# EPICS autosave request: autosave/galil_motors.req
$(P)$(M)_able
$(P)$(M)Direction
$(P)$(M)Offset
$(P)$(M)Resolution
$(P)$(M)_PCOF_SP
$(P)$(M)_ICOF_SP
$(P)$(M)_DCOF_SP
$(P)$(M)_ACCL_SP
$(P)$(M)_RDBD_SP
$(P)$(M)_VMAX_SP
$(P)$(M)_VELO_SP
$(P)$(M)_OFF_SP
$(P)$(M)_MRES_SP
$(P)$(M)_ERES_SP
$(P)$(M)_DIR_SP
$(P)$(M)_DMOV_SP
$(P)$(M)_SET_SP
$(P)$(M)_UEIP_SP
$(P)$(M)_SPMG_SP
$(P)$(M)_PREM_CMD
$(P)$(M)_POST_CMD
# $(P)$(M)_STOPGO_CMD
$(P)$(M)_VALOUT_SP
$(P)$(M).ACCL
$(P)$(M).ADEL
$(P)$(M).BACC
$(P)$(M).BDST
$(P)$(M).BVEL
$(P)$(M).CNEN
$(P)$(M).DCOF
$(P)$(M).DHLM
$(P)$(M).DINP
$(P)$(M).DIR
$(P)$(M).DLLM
$(P)$(M).DLY
$(P)$(M).DVAL
$(P)$(M).EGU
$(P)$(M).ERES
$(P)$(M).FOF
$(P)$(M).FOFF
$(P)$(M).FRAC
$(P)$(M).HHSV
$(P)$(M).HIGH
$(P)$(M).HIHI
$(P)$(M).HLM
$(P)$(M).HLSV
$(P)$(M).RDBL

$(P)$(M).HOMF
$(P)$(M).HOMR
$(P)$(M).HOPR
$(P)$(M).HSV
$(P)$(M).HVEL
$(P)$(M).ICOF
$(P)$(M).IGSET
$(P)$(M).INIT
$(P)$(M).JAR
$(P)$(M).JOGR
$(P)$(M).JOGF
$(P)$(M).JVEL
$(P)$(M).LLM
$(P)$(M).LLSV
$(P)$(M).LOCK
$(P)$(M).LOLO
$(P)$(M).LOPR
$(P)$(M).LOW
$(P)$(M).LSV
$(P)$(M).MDEL
$(P)$(M).NTM
$(P)$(M).NTMF
$(P)$(M).OFF
$(P)$(M).OMSL
$(P)$(M).OUT
$(P)$(M).PCOF
$(P)$(M).POST
$(P)$(M).PREC
$(P)$(M).PREM
$(P)$(M).RDBD
$(P)$(M).RINP
$(P)$(M).RLV
$(P)$(M).RMOD
$(P)$(M).RRES
$(P)$(M).RTRY
$(P)$(M).RVAL
$(P)$(M).S
$(P)$(M).SBAK
$(P)$(M).SBAS
$(P)$(M).SET
$(P)$(M).SMAX
$(P)$(M).SPMG
$(P)$(M).SREV
$(P)$(M).SSET
$(P)$(M).STOO
$(P)$(M).STOP
$(P)$(M).STUP
$(P)$(M).SUSE
$(P)$(M).SYNC
$(P)$(M).TWF
$(P)$(M).TWR
$(P)$(M).TWV
$(P)$(M).UEIP
$(P)$(M).UREV
$(P)$(M).URIP
$(P)$(M).VBAS
$(P)$(M).VELO
$(P)$(M).VMAX
$(P)$(M).VOF
